FUNCTION_BLOCK FB_ST10b
VAR
	_test : BOOL; 
END_VAR

METHOD _test : BOOL
VAR_INPUT
END_VAR
_test:= TRUE;
END_METHOD

END_FUNCTION_BLOCK

(* stored: Version 1.1.0.1, ProductVersion 3.1.4024.12
   POU FB_ST10b: Id {6ce20a51-ab97-4003-969b-df3949d611fe}, SpecialFunc None
   Method _test: Id {41f4d043-bc9c-467f-be6d-604ea26985e1} *)
